PROGRAM AxisMoveAbsoulte
VAR
END_VAR

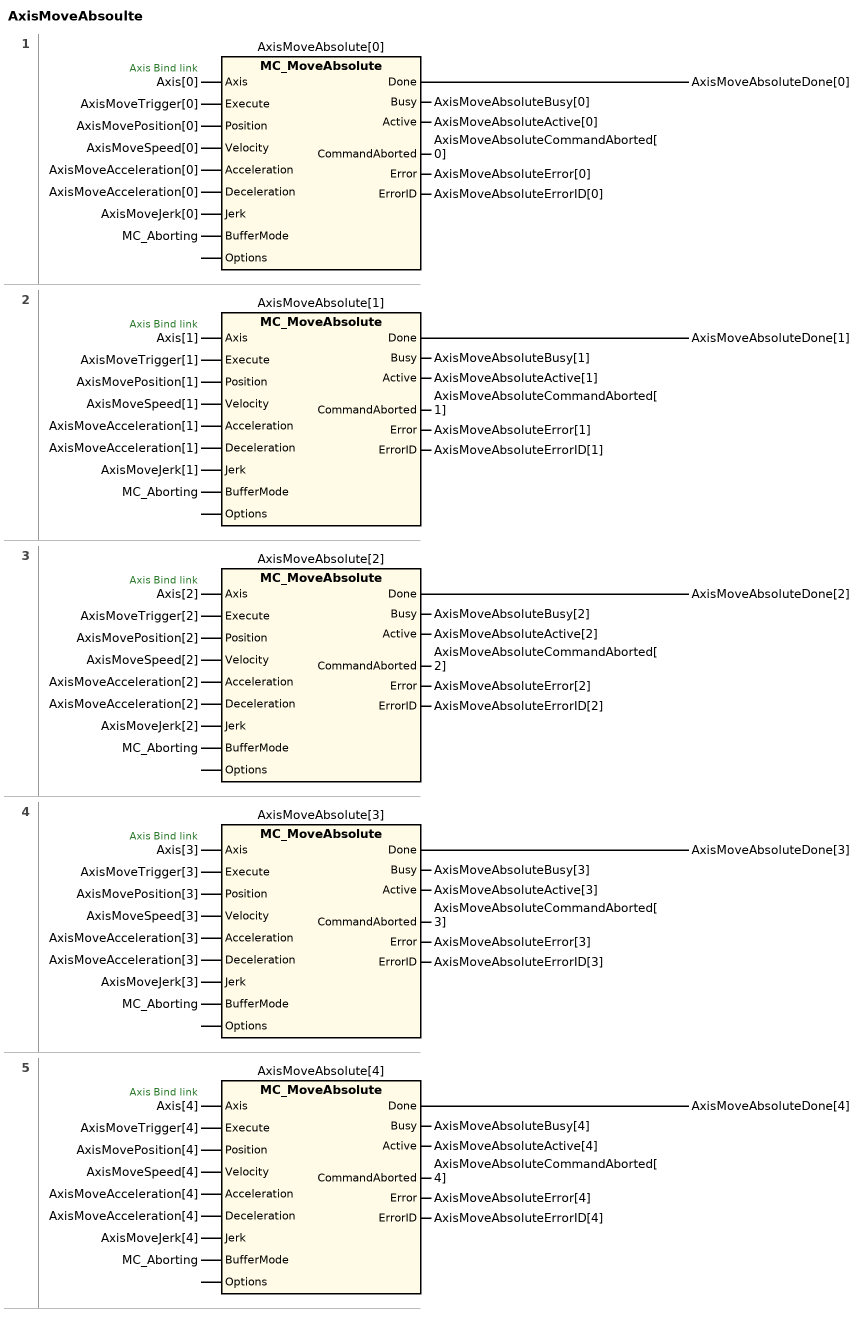
// NETWORK 1
//   AxisMoveAbsolute[0]: Axis Move Absolute
//   Axis[0]: Axis Bind link
AxisMoveAbsolute[0](
    Axis := Axis[0],
    Execute := AxisMoveTrigger[0],
    Position := AxisMovePosition[0],
    Velocity := AxisMoveSpeed[0],
    Acceleration := AxisMoveAcceleration[0],
    Deceleration := AxisMoveAcceleration[0],
    Jerk := AxisMoveJerk[0],
    BufferMode := MC_Aborting,
    Busy => AxisMoveAbsoluteBusy[0],
    Active => AxisMoveAbsoluteActive[0],
    CommandAborted => AxisMoveAbsoluteCommandAborted[0],
    Error => AxisMoveAbsoluteError[0],
    ErrorID => AxisMoveAbsoluteErrorID[0]); // MC_MoveAbsolute
AxisMoveAbsoluteDone[0] := AxisMoveAbsolute[0].Done;

// NETWORK 2
//   AxisMoveAbsolute[1]: Axis Move Absolute
//   Axis[1]: Axis Bind link
AxisMoveAbsolute[1](
    Axis := Axis[1],
    Execute := AxisMoveTrigger[1],
    Position := AxisMovePosition[1],
    Velocity := AxisMoveSpeed[1],
    Acceleration := AxisMoveAcceleration[1],
    Deceleration := AxisMoveAcceleration[1],
    Jerk := AxisMoveJerk[1],
    BufferMode := MC_Aborting,
    Busy => AxisMoveAbsoluteBusy[1],
    Active => AxisMoveAbsoluteActive[1],
    CommandAborted => AxisMoveAbsoluteCommandAborted[1],
    Error => AxisMoveAbsoluteError[1],
    ErrorID => AxisMoveAbsoluteErrorID[1]); // MC_MoveAbsolute
AxisMoveAbsoluteDone[1] := AxisMoveAbsolute[1].Done;

// NETWORK 3
//   AxisMoveAbsolute[2]: Axis Move Absolute
//   Axis[2]: Axis Bind link
AxisMoveAbsolute[2](
    Axis := Axis[2],
    Execute := AxisMoveTrigger[2],
    Position := AxisMovePosition[2],
    Velocity := AxisMoveSpeed[2],
    Acceleration := AxisMoveAcceleration[2],
    Deceleration := AxisMoveAcceleration[2],
    Jerk := AxisMoveJerk[2],
    BufferMode := MC_Aborting,
    Busy => AxisMoveAbsoluteBusy[2],
    Active => AxisMoveAbsoluteActive[2],
    CommandAborted => AxisMoveAbsoluteCommandAborted[2],
    Error => AxisMoveAbsoluteError[2],
    ErrorID => AxisMoveAbsoluteErrorID[2]); // MC_MoveAbsolute
AxisMoveAbsoluteDone[2] := AxisMoveAbsolute[2].Done;

// NETWORK 4
//   AxisMoveAbsolute[3]: Axis Move Absolute
//   Axis[3]: Axis Bind link
AxisMoveAbsolute[3](
    Axis := Axis[3],
    Execute := AxisMoveTrigger[3],
    Position := AxisMovePosition[3],
    Velocity := AxisMoveSpeed[3],
    Acceleration := AxisMoveAcceleration[3],
    Deceleration := AxisMoveAcceleration[3],
    Jerk := AxisMoveJerk[3],
    BufferMode := MC_Aborting,
    Busy => AxisMoveAbsoluteBusy[3],
    Active => AxisMoveAbsoluteActive[3],
    CommandAborted => AxisMoveAbsoluteCommandAborted[3],
    Error => AxisMoveAbsoluteError[3],
    ErrorID => AxisMoveAbsoluteErrorID[3]); // MC_MoveAbsolute
AxisMoveAbsoluteDone[3] := AxisMoveAbsolute[3].Done;

// NETWORK 5
//   AxisMoveAbsolute[4]: Axis Move Absolute
//   Axis[4]: Axis Bind link
AxisMoveAbsolute[4](
    Axis := Axis[4],
    Execute := AxisMoveTrigger[4],
    Position := AxisMovePosition[4],
    Velocity := AxisMoveSpeed[4],
    Acceleration := AxisMoveAcceleration[4],
    Deceleration := AxisMoveAcceleration[4],
    Jerk := AxisMoveJerk[4],
    BufferMode := MC_Aborting,
    Busy => AxisMoveAbsoluteBusy[4],
    Active => AxisMoveAbsoluteActive[4],
    CommandAborted => AxisMoveAbsoluteCommandAborted[4],
    Error => AxisMoveAbsoluteError[4],
    ErrorID => AxisMoveAbsoluteErrorID[4]); // MC_MoveAbsolute
AxisMoveAbsoluteDone[4] := AxisMoveAbsolute[4].Done;

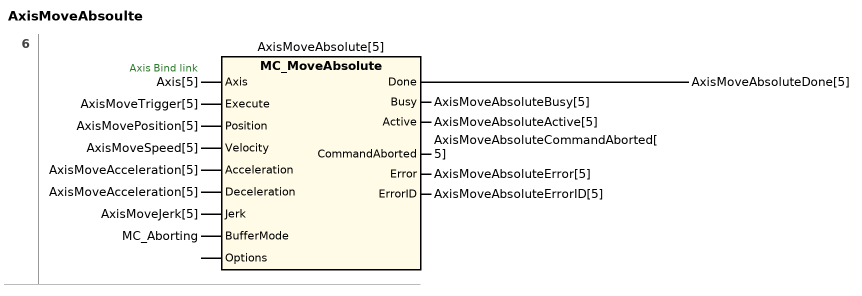
// NETWORK 6
//   AxisMoveAbsolute[5]: Axis Move Absolute
//   Axis[5]: Axis Bind link
AxisMoveAbsolute[5](
    Axis := Axis[5],
    Execute := AxisMoveTrigger[5],
    Position := AxisMovePosition[5],
    Velocity := AxisMoveSpeed[5],
    Acceleration := AxisMoveAcceleration[5],
    Deceleration := AxisMoveAcceleration[5],
    Jerk := AxisMoveJerk[5],
    BufferMode := MC_Aborting,
    Busy => AxisMoveAbsoluteBusy[5],
    Active => AxisMoveAbsoluteActive[5],
    CommandAborted => AxisMoveAbsoluteCommandAborted[5],
    Error => AxisMoveAbsoluteError[5],
    ErrorID => AxisMoveAbsoluteErrorID[5]); // MC_MoveAbsolute
AxisMoveAbsoluteDone[5] := AxisMoveAbsolute[5].Done;

END_PROGRAM

(* stored: Version 1.1.0.1, ProductVersion 3.1.4018.5
   POU AxisMoveAbsoulte: Id {07268d8a-f4aa-4667-b584-ad3731dd61a3}, SpecialFunc None *)
